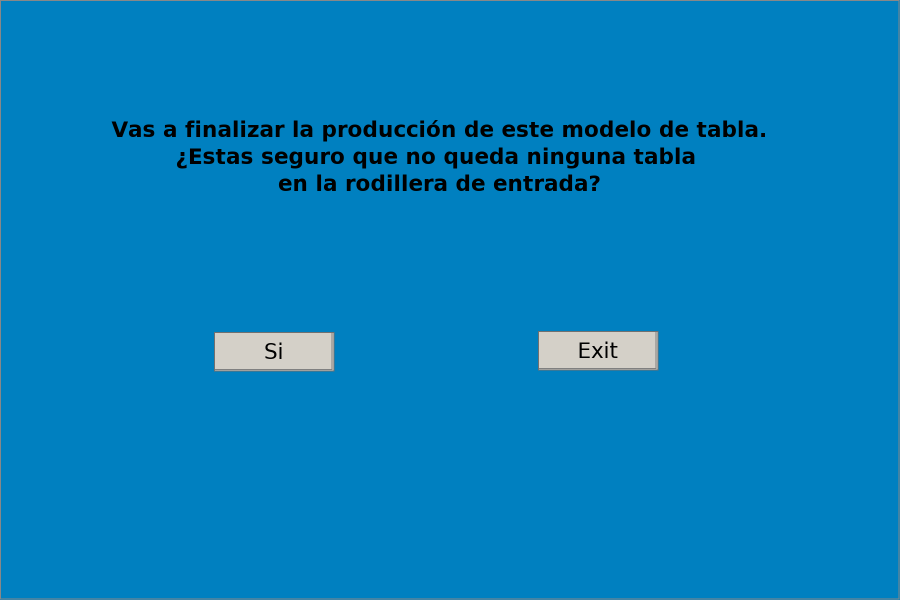
VISUALIZATION V_Emerg_Fin_Prod_Md1  // 900x600
    Button (214,332 120x39), "Si"
        tap FuncParoNodoMultidiscos.FunGeneMultidiscos1.P_FinProduccion p3779583253=TRUE
        OnMouseClick: change screen: Modelo_Tabla_Md1
        OnMouseClick: CloseDialog Dialog=V_Emerg_Fin_Prod_Md1, Result=OK, NumpadKeypadSet=True
    Button (538,331 120x39), "Exit"
        OnMouseClick: CloseDialog Dialog=V_Emerg_Fin_Prod_Ch4, Result=OK, NumpadKeypadSet=True
    Label (113,67 653x179), "Vas a finalizar la producción de este modelo de tabla. ¿Estas seguro que no queda ninguna tabla en la rodillera de entrada?"
END_VISUALIZATION

(* stored: Version 1.1.0.1, ProductVersion 3.1.4024.12
   Visu V_Emerg_Fin_Prod_Md1: Id {56a9b5bd-e06b-48e3-bec6-57d595adc171} *)
